% RSLogix 500 project I2P Job 11 - Tyler_Vogt.RSS, saved by version 10.00.00.00 %
PROJECT "MLO2B"    % processor: Bul.1763 MicroLogix 1100 Series B %

PROGRAM FILES
  LAD 2   6 rungs

DATA FILES
  O0 OUTPUT  4 elements
  I1 INPUT  6 elements
  S2 STATUS  66 elements
  B3 BINARY  1 elements
  T4 TIMER  1 elements
  C5 COUNTER  1 elements
  R6 CONTROL  1 elements
  N7 INTEGER  1 elements
  F8 FLOAT  1 elements

LADDER 2
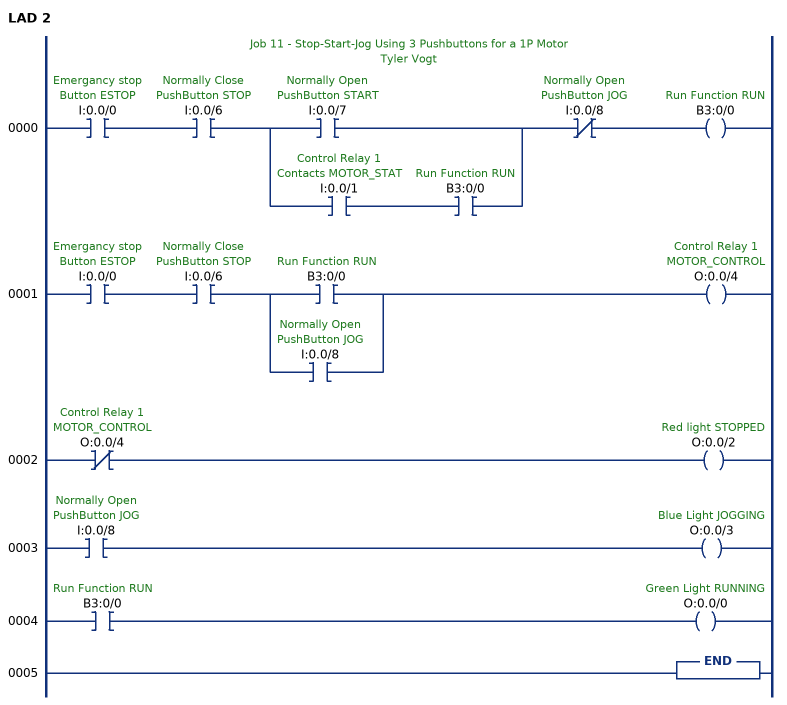
% Rung: 0 %
% Job 11 - Stop-Start-Jog Using 3 Pushbuttons for a 1P Motor
% Tyler Vogt %
SOR XIC I:0.0/0 XIC I:0.0/6 BST XIC I:0.0/7 NXB XIC I:0.0/1 XIC B3:0/0 BND XIO I:0.0/8 OTE B3:0/0 EOR
%   I:0.0/0  ESTOP  "Emergancy stop Button" %
%   I:0.0/6  STOP  "Normally Close PushButton" %
%   I:0.0/7  START  "Normally Open PushButton" %
%   I:0.0/1  MOTOR_STAT  "Control Relay 1 Contacts" %
%   B3:0/0  RUN  "Run Function" %
%   I:0.0/8  JOG  "Normally Open PushButton" %
% Rung: 1 %
SOR XIC I:0.0/0 XIC I:0.0/6 BST XIC B3:0/0 NXB XIC I:0.0/8 BND OTE O:0.0/4 EOR
%   I:0.0/0  ESTOP  "Emergancy stop Button" %
%   I:0.0/6  STOP  "Normally Close PushButton" %
%   B3:0/0  RUN  "Run Function" %
%   I:0.0/8  JOG  "Normally Open PushButton" %
%   O:0.0/4  MOTOR_CONTROL  "Control Relay 1" %
% Rung: 2 %
SOR XIO O:0.0/4 OTE O:0.0/2 EOR
%   O:0.0/4  MOTOR_CONTROL  "Control Relay 1" %
%   O:0.0/2  STOPPED  "Red light" %
% Rung: 3 %
SOR XIC I:0.0/8 OTE O:0.0/3 EOR
%   I:0.0/8  JOG  "Normally Open PushButton" %
%   O:0.0/3  JOGGING  "Blue Light" %
% Rung: 4 %
SOR XIC B3:0/0 OTE O:0.0/0 EOR
%   B3:0/0  RUN  "Run Function" %
%   O:0.0/0  RUNNING  "Green Light" %
% Rung: 5 %
SOR END EOR

OTHER DOCUMENTED ADDRESSES
  I:0.0/2  CR2_STAT  "Control Relay 2 Contacts"
  I:0.0/3  3PSS_A  "3 Position Selector Switch A Position"
  I:0.0/4  3PSS_B  "3 Position Selector Switch B Position"
  I:0.0/5  RUN_JOG  "2 Position Selector Switch A Position"
  O:0.0/1  YLW_LT  "Yellow Light"
  O:0.0/5  CR2  "Control Relay 2"
